PROGRAM PRG_LARS_ValidationAsConfirmation_ORG
VAR
	rtrigNewOuterArrived					: R_TRIG;
	bNewOuterIsProccesing				: BOOL;
	tonValidationTimout					: TON;
	bValidationTimeout					: BOOL;
	bValidationTimeoutReset				: BOOL;
	fbTimeoutCounter						: CTU;
	nCount									: INT;
	fbPerformance							: FB_Interval;

	fbOuterValidationCamera				: FB_SCANNER_CameraSelect;
	(*stOuterValidationCameraOptions		: ST_SCANNER_Options := (eScannerType := E_MV_420_FULL, nImageBuffer := 1, nExpectedResp := 2);*)
	fbOuterValidationEvaluation			: FB_SCANNER_Evaluation;

	fbCheckForDuplicateOuterValidation	: FB_OUTER_CheckDuplicateStatus;

	rtrigOuterValidationCameraDone		: R_TRIG;
	bOuterValidationCameraDone			: BOOL;
	bDataReadyForValidation				: BOOL;
	bQAReject								: BOOL;

	sLastImageLableString				: T_OUTER_Barcode;

	fbMoveOuterData						: FB_OUTER_MoveOuterStatus;
	fbCompleteDataFromConfirmation	: FB_OUTER_CompleteDataFromConfirmation;
	fbMETSValidateOuterForReject			: FB_OUTER_ValidateOuterForReject;
	tofValidateOuterDoneForHMI			: TOF;
	fbMasterListUpdate					: FB_OUTER_MasterListUpdate;

	stLastOuterCompleted					: ST_OUTER_Status;
	sLastReadOuterBarcode				: T_OUTER_Barcode;
	sLastReadConfPackCode1				: T_PACK_Barcode;
	nOutersCompleted						: UDINT;
	bDoneInfo								: BOOL;

	rtrigSetOuterValidationOK			: R_TRIG;
	rtrigSetOuterValidationNOK		: R_TRIG;

	rsOuterRejectStation 				: RS;
	rsOuterRejectConfirmation 		: RS;

	rtrigResetValidationStatus			: R_TRIG;

	sRejectCode						: STRING(255);
	fbArchiveInvalidOuters			: FB_OUTER_ArchiveInvalidOuters;
	aReasonForReject					: ARRAY[0..50] OF STRING(255);
	bClearList							: BOOL;

	fbOuterProduced					: FB_KPI_GenericEfficiency;
	fbOuterInspection					: FB_KPI_OutersEfficiency;

	fbOuterLevelCounter				: FB_KPI_OuterLevelCounter;

	fbQARejectCounter				: FB_CTU32;
	fbOuterValidationIndexOK			: FB_CTU32;

	ctuConsecutiveOuterRejects		: CTU;
	nActualCount						: INT;

	stDummyImageData			: ST_SCANNER_ImageData;		(* image data structure *)
	aDistanceCheck				: ARRAY[1..2] OF FB_TimeDistance;
	bResetCTU						: BOOL;
END_VAR
VAR // added by the converter: edge detectors and wires of the graphical bodies
    _w1 : BOOL;
END_VAR

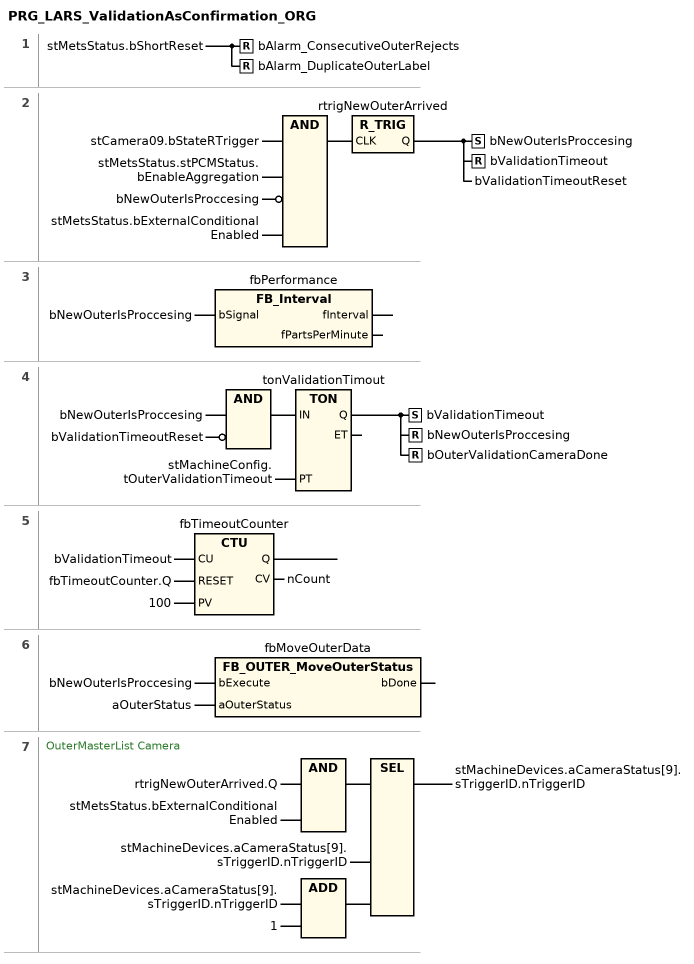
// NETWORK 1
bAlarm_ConsecutiveOuterRejects R= stMetsStatus.bShortReset;
bAlarm_DuplicateOuterLabel R= stMetsStatus.bShortReset;

// NETWORK 2
rtrigNewOuterArrived(CLK := stCamera09.bStateRTrigger AND stMetsStatus.stPCMStatus.bEnableAggregation AND NOT bNewOuterIsProccesing AND stMetsStatus.bExternalConditionalEnabled); // R_TRIG
bNewOuterIsProccesing S= rtrigNewOuterArrived.Q;
bValidationTimeout R= rtrigNewOuterArrived.Q;
bValidationTimeoutReset := rtrigNewOuterArrived.Q;

// NETWORK 3
fbPerformance(bSignal := bNewOuterIsProccesing); // FB_Interval

// NETWORK 4
tonValidationTimout(IN := bNewOuterIsProccesing AND NOT bValidationTimeoutReset, PT := stMachineConfig.tOuterValidationTimeout); // TON
bValidationTimeout S= tonValidationTimout.Q;
bNewOuterIsProccesing R= tonValidationTimout.Q;
bOuterValidationCameraDone R= tonValidationTimout.Q;

// NETWORK 5
fbTimeoutCounter(CU := bValidationTimeout, RESET := fbTimeoutCounter.Q, PV := 100, CV => nCount); // CTU

// NETWORK 6
fbMoveOuterData(bExecute := bNewOuterIsProccesing, aOuterStatus := aOuterStatus); // FB_OUTER_MoveOuterStatus

// NETWORK 7
// OuterMasterList Camera
stMachineDevices.aCameraStatus[9].sTriggerID.nTriggerID := SEL(rtrigNewOuterArrived.Q AND stMetsStatus.bExternalConditionalEnabled, stMachineDevices.aCameraStatus[9].sTriggerID.nTriggerID, stMachineDevices.aCameraStatus[9].sTriggerID.nTriggerID + 1);

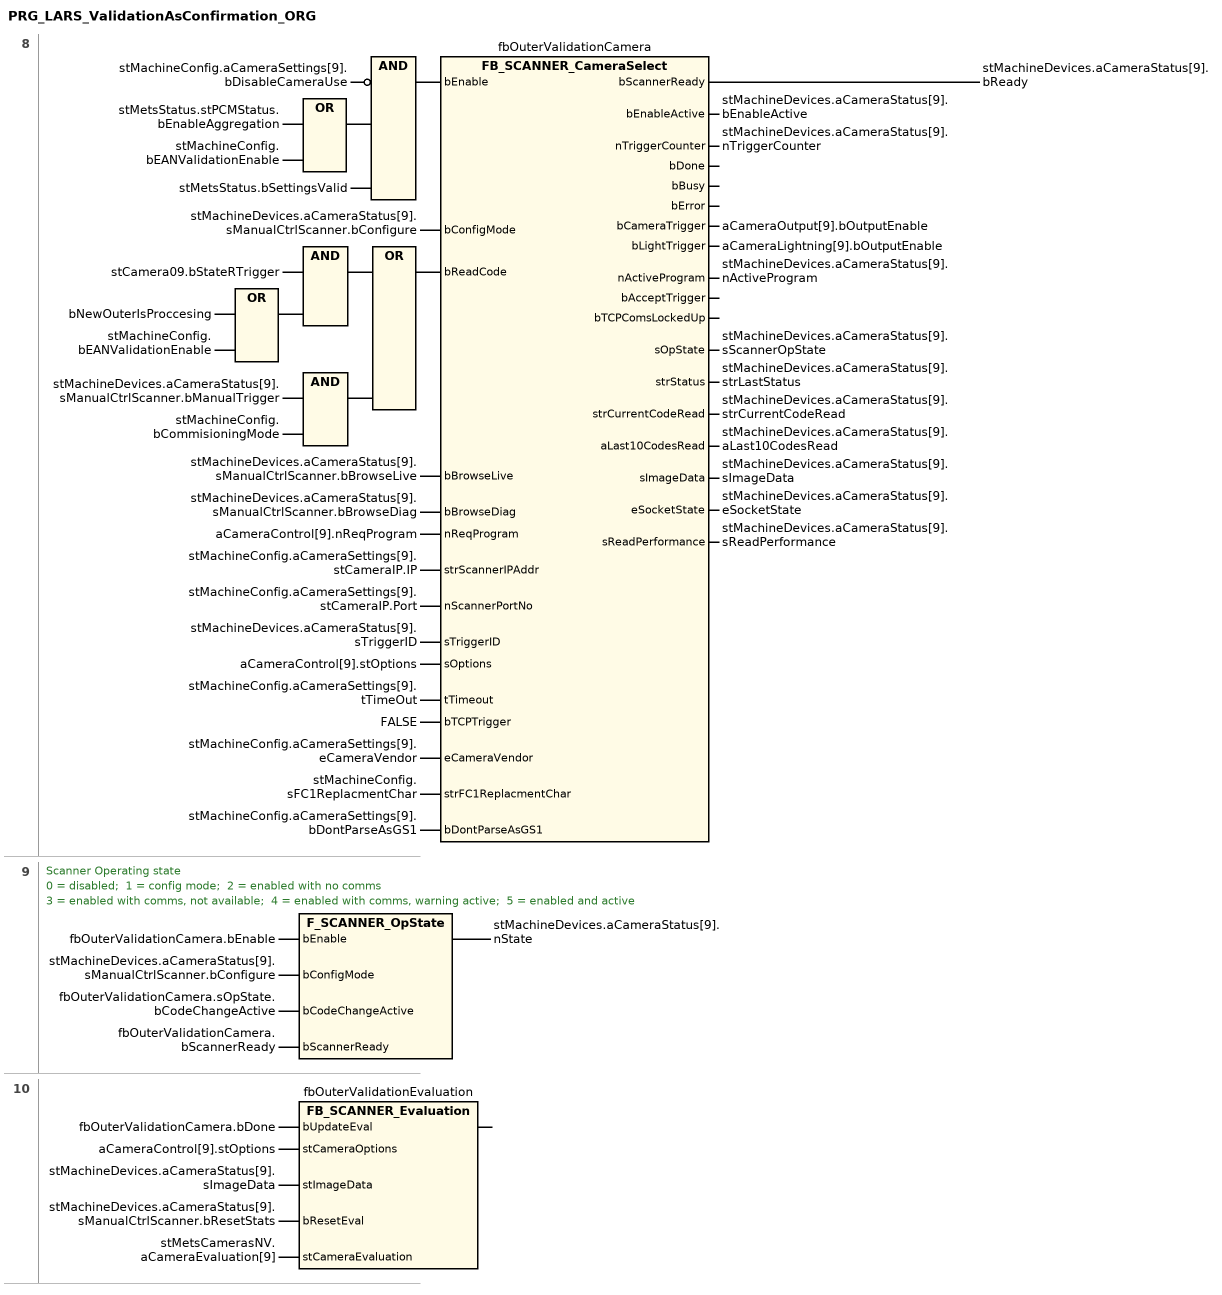
// NETWORK 8
fbOuterValidationCamera(
    bEnable := NOT stMachineConfig.aCameraSettings[9].bDisableCameraUse AND (stMetsStatus.stPCMStatus.bEnableAggregation OR stMachineConfig.bEANValidationEnable) AND stMetsStatus.bSettingsValid,
    bConfigMode := stMachineDevices.aCameraStatus[9].sManualCtrlScanner.bConfigure,
    bReadCode := stCamera09.bStateRTrigger AND (bNewOuterIsProccesing OR stMachineConfig.bEANValidationEnable) OR stMachineDevices.aCameraStatus[9].sManualCtrlScanner.bManualTrigger AND stMachineConfig.bCommisioningMode,
    bBrowseLive := stMachineDevices.aCameraStatus[9].sManualCtrlScanner.bBrowseLive,
    bBrowseDiag := stMachineDevices.aCameraStatus[9].sManualCtrlScanner.bBrowseDiag,
    nReqProgram := aCameraControl[9].nReqProgram,
    strScannerIPAddr := stMachineConfig.aCameraSettings[9].stCameraIP.IP,
    nScannerPortNo := stMachineConfig.aCameraSettings[9].stCameraIP.Port,
    sTriggerID := stMachineDevices.aCameraStatus[9].sTriggerID,
    sOptions := aCameraControl[9].stOptions,
    tTimeout := stMachineConfig.aCameraSettings[9].tTimeOut,
    bTCPTrigger := FALSE,
    eCameraVendor := stMachineConfig.aCameraSettings[9].eCameraVendor,
    strFC1ReplacmentChar := stMachineConfig.sFC1ReplacmentChar,
    bDontParseAsGS1 := stMachineConfig.aCameraSettings[9].bDontParseAsGS1,
    bEnableActive => stMachineDevices.aCameraStatus[9].bEnableActive,
    nTriggerCounter => stMachineDevices.aCameraStatus[9].nTriggerCounter,
    bCameraTrigger => aCameraOutput[9].bOutputEnable,
    bLightTrigger => aCameraLightning[9].bOutputEnable,
    nActiveProgram => stMachineDevices.aCameraStatus[9].nActiveProgram,
    sOpState => stMachineDevices.aCameraStatus[9].sScannerOpState,
    strStatus => stMachineDevices.aCameraStatus[9].strLastStatus,
    strCurrentCodeRead => stMachineDevices.aCameraStatus[9].strCurrentCodeRead,
    aLast10CodesRead => stMachineDevices.aCameraStatus[9].aLast10CodesRead,
    sImageData => stMachineDevices.aCameraStatus[9].sImageData,
    eSocketState => stMachineDevices.aCameraStatus[9].eSocketState,
    sReadPerformance => stMachineDevices.aCameraStatus[9].sReadPerformance); // FB_SCANNER_CameraSelect
stMachineDevices.aCameraStatus[9].bReady := fbOuterValidationCamera.bScannerReady;

// NETWORK 9
// 					Scanner Operating state
// 0 = disabled;  1 = config mode;  2 = enabled with no comms
// 3 = enabled with comms, not available;  4 = enabled with comms, warning active;  5 = enabled and active
//
stMachineDevices.aCameraStatus[9].nState := F_SCANNER_OpState(bEnable := fbOuterValidationCamera.bEnable, bConfigMode := stMachineDevices.aCameraStatus[9].sManualCtrlScanner.bConfigure, bCodeChangeActive := fbOuterValidationCamera.sOpState.bCodeChangeActive, bScannerReady := fbOuterValidationCamera.bScannerReady);

// NETWORK 10
fbOuterValidationEvaluation(
    bUpdateEval := fbOuterValidationCamera.bDone,
    stCameraOptions := aCameraControl[9].stOptions,
    stImageData := stMachineDevices.aCameraStatus[9].sImageData,
    bResetEval := stMachineDevices.aCameraStatus[9].sManualCtrlScanner.bResetStats,
    stCameraEvaluation := stMetsCamerasNV.aCameraEvaluation[9]); // FB_SCANNER_Evaluation

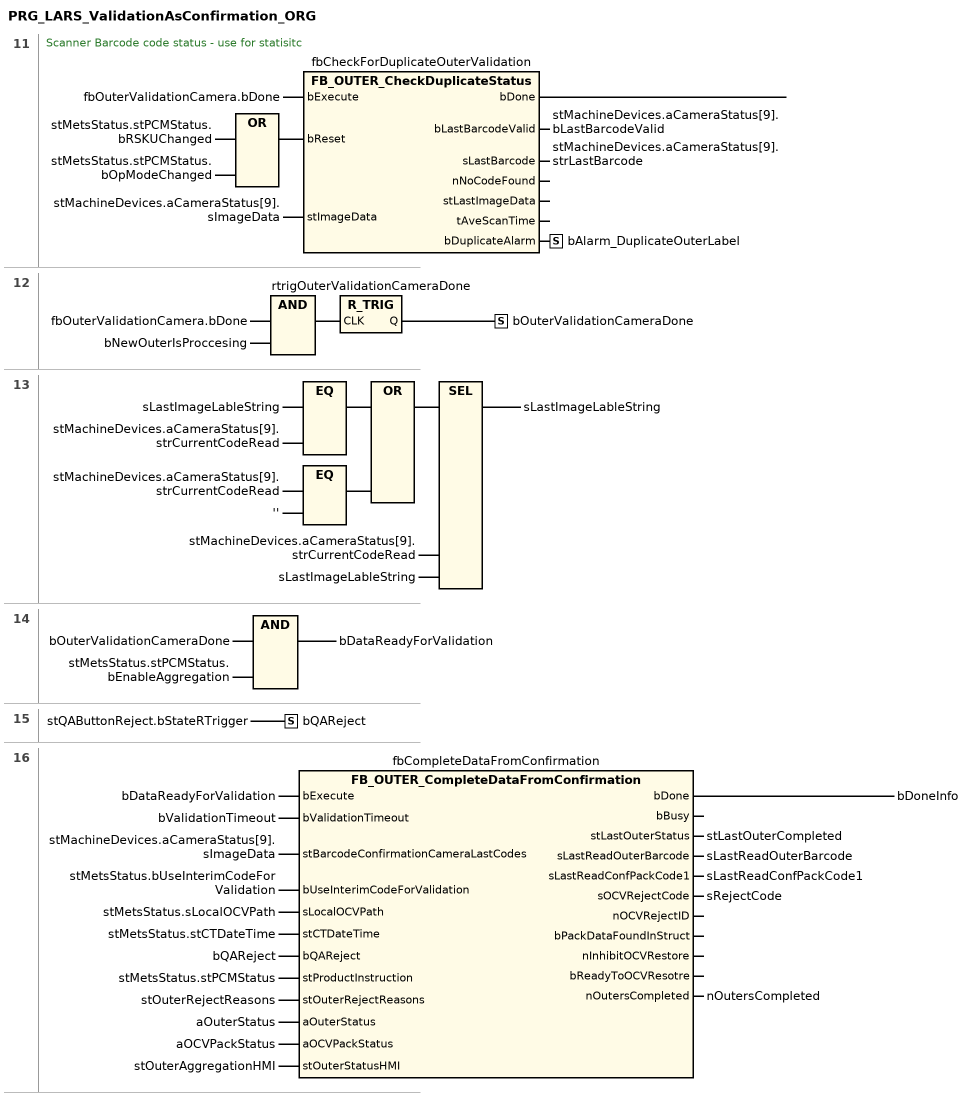
// NETWORK 11
// Scanner Barcode code status - use for statisitc
fbCheckForDuplicateOuterValidation(
    bExecute := fbOuterValidationCamera.bDone,
    bReset := stMetsStatus.stPCMStatus.bRSKUChanged OR stMetsStatus.stPCMStatus.bOpModeChanged,
    stImageData := stMachineDevices.aCameraStatus[9].sImageData,
    bLastBarcodeValid => stMachineDevices.aCameraStatus[9].bLastBarcodeValid,
    sLastBarcode => stMachineDevices.aCameraStatus[9].strLastBarcode); // FB_OUTER_CheckDuplicateStatus
bAlarm_DuplicateOuterLabel S= fbCheckForDuplicateOuterValidation.bDuplicateAlarm;

// NETWORK 12
rtrigOuterValidationCameraDone(CLK := fbOuterValidationCamera.bDone AND bNewOuterIsProccesing); // R_TRIG
bOuterValidationCameraDone S= rtrigOuterValidationCameraDone.Q;

// NETWORK 13
sLastImageLableString := SEL(sLastImageLableString = stMachineDevices.aCameraStatus[9].strCurrentCodeRead OR stMachineDevices.aCameraStatus[9].strCurrentCodeRead = '', stMachineDevices.aCameraStatus[9].strCurrentCodeRead, sLastImageLableString);

// NETWORK 14
bDataReadyForValidation := bOuterValidationCameraDone AND stMetsStatus.stPCMStatus.bEnableAggregation;

// NETWORK 15
bQAReject S= stQAButtonReject.bStateRTrigger;

// NETWORK 16
fbCompleteDataFromConfirmation(
    bExecute := bDataReadyForValidation,
    bValidationTimeout := bValidationTimeout,
    stBarcodeConfirmationCameraLastCodes := stMachineDevices.aCameraStatus[9].sImageData,
    bUseInterimCodeForValidation := stMetsStatus.bUseInterimCodeForValidation,
    sLocalOCVPath := stMetsStatus.sLocalOCVPath,
    stCTDateTime := stMetsStatus.stCTDateTime,
    bQAReject := bQAReject,
    stProductInstruction := stMetsStatus.stPCMStatus,
    stOuterRejectReasons := stOuterRejectReasons,
    aOuterStatus := aOuterStatus,
    aOCVPackStatus := aOCVPackStatus,
    stOuterStatusHMI := stOuterAggregationHMI,
    stLastOuterStatus => stLastOuterCompleted,
    sLastReadOuterBarcode => sLastReadOuterBarcode,
    sLastReadConfPackCode1 => sLastReadConfPackCode1,
    sOCVRejectCode => sRejectCode,
    nOutersCompleted => nOutersCompleted); // FB_OUTER_CompleteDataFromConfirmation
bDoneInfo := fbCompleteDataFromConfirmation.bDone;

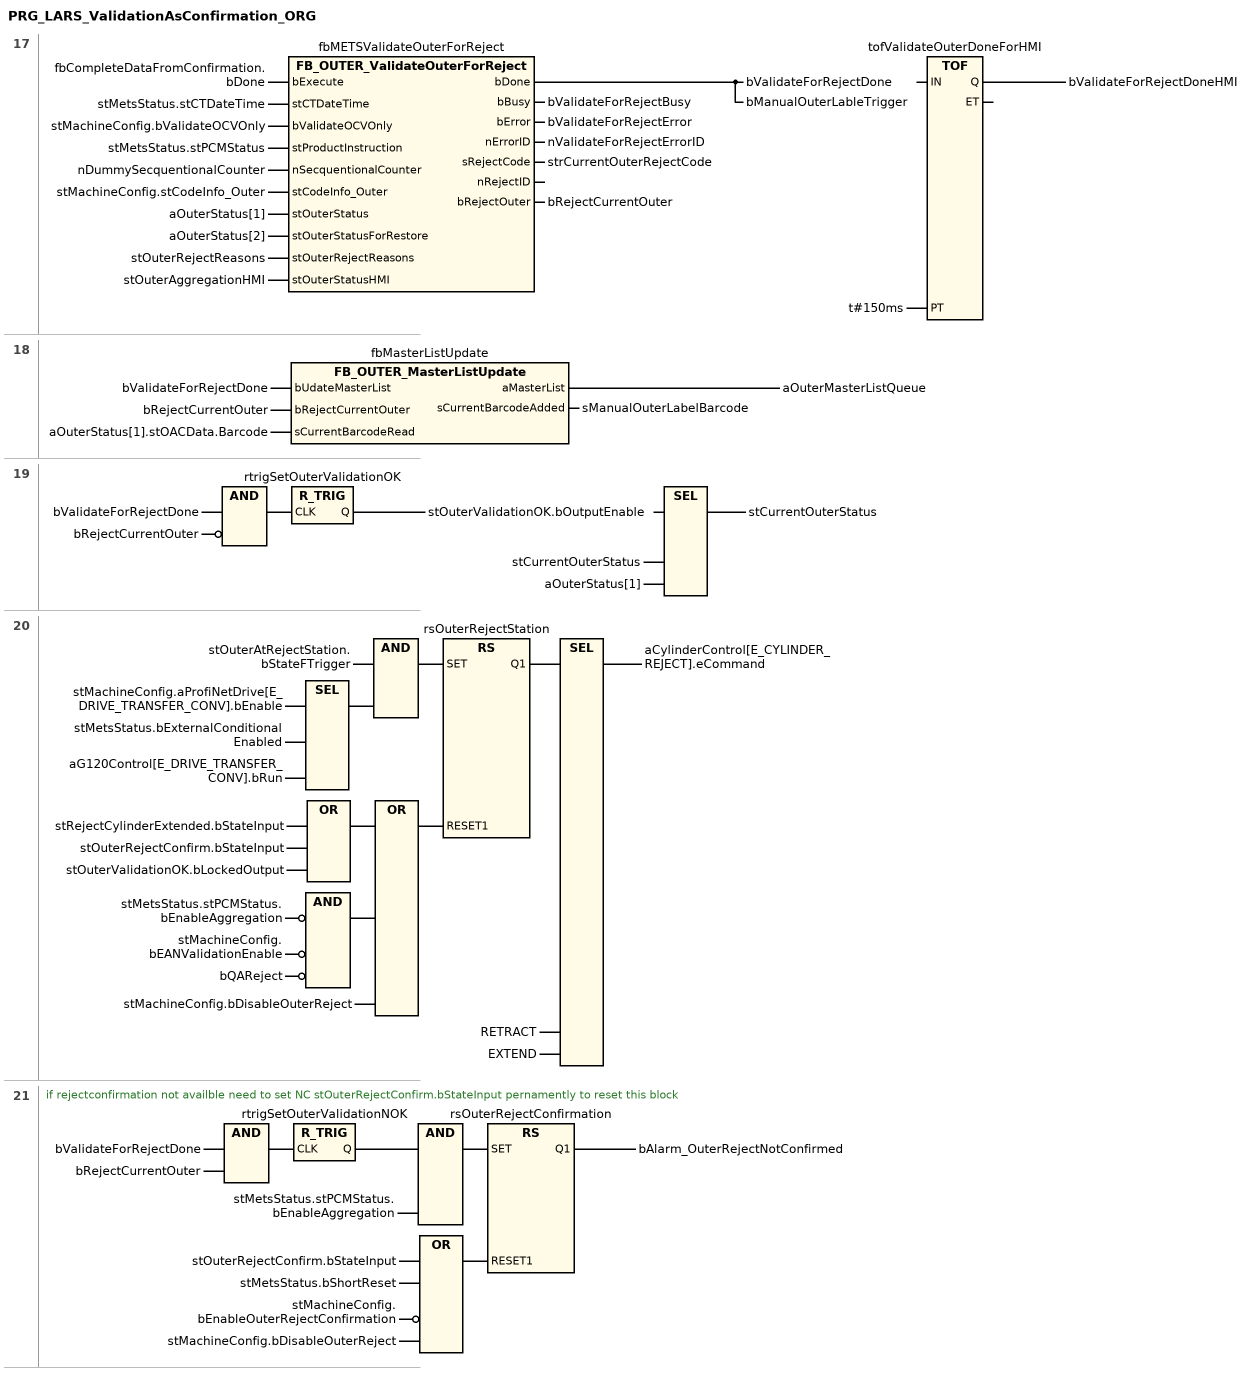
// NETWORK 17
fbMETSValidateOuterForReject(
    bExecute := fbCompleteDataFromConfirmation.bDone,
    stCTDateTime := stMetsStatus.stCTDateTime,
    bValidateOCVOnly := stMachineConfig.bValidateOCVOnly,
    stProductInstruction := stMetsStatus.stPCMStatus,
    nSecquentionalCounter := nDummySecquentionalCounter,
    stCodeInfo_Outer := stMachineConfig.stCodeInfo_Outer,
    stOuterStatus := aOuterStatus[1],
    stOuterStatusForRestore := aOuterStatus[2],
    stOuterRejectReasons := stOuterRejectReasons,
    stOuterStatusHMI := stOuterAggregationHMI,
    bBusy => bValidateForRejectBusy,
    bError => bValidateForRejectError,
    nErrorID => nValidateForRejectErrorID,
    sRejectCode => strCurrentOuterRejectCode,
    bRejectOuter => bRejectCurrentOuter); // FB_OUTER_ValidateOuterForReject
bValidateForRejectDone := fbMETSValidateOuterForReject.bDone;
bManualOuterLableTrigger := fbMETSValidateOuterForReject.bDone;
tofValidateOuterDoneForHMI(IN := fbMETSValidateOuterForReject.bDone, PT := t#150ms); // TOF
bValidateForRejectDoneHMI := tofValidateOuterDoneForHMI.Q;

// NETWORK 18
fbMasterListUpdate(
    bUdateMasterList := bValidateForRejectDone,
    bRejectCurrentOuter := bRejectCurrentOuter,
    sCurrentBarcodeRead := aOuterStatus[1].stOACData.Barcode,
    sCurrentBarcodeAdded => sManualOuterLabelBarcode); // FB_OUTER_MasterListUpdate
aOuterMasterListQueue := fbMasterListUpdate.aMasterList;

// NETWORK 19
rtrigSetOuterValidationOK(CLK := bValidateForRejectDone AND NOT bRejectCurrentOuter); // R_TRIG
stOuterValidationOK.bOutputEnable := rtrigSetOuterValidationOK.Q;
stCurrentOuterStatus := SEL(rtrigSetOuterValidationOK.Q, stCurrentOuterStatus, aOuterStatus[1]);

// NETWORK 20
rsOuterRejectStation(SET := stOuterAtRejectStation.bStateFTrigger AND SEL(stMachineConfig.aProfiNetDrive[E_DRIVE_TRANSFER_CONV].bEnable, stMetsStatus.bExternalConditionalEnabled, aG120Control[E_DRIVE_TRANSFER_CONV].bRun), RESET1 := (stRejectCylinderExtended.bStateInput OR stOuterRejectConfirm.bStateInput OR stOuterValidationOK.bLockedOutput) OR NOT stMetsStatus.stPCMStatus.bEnableAggregation AND NOT stMachineConfig.bEANValidationEnable AND NOT bQAReject OR stMachineConfig.bDisableOuterReject); // RS
aCylinderControl[E_CYLINDER_REJECT].eCommand := SEL(rsOuterRejectStation.Q1, RETRACT, EXTEND);

// NETWORK 21
// if rejectconfirmation not availble need to set NC stOuterRejectConfirm.bStateInput pernamently to reset this block
rtrigSetOuterValidationNOK(CLK := bValidateForRejectDone AND bRejectCurrentOuter); // R_TRIG
rsOuterRejectConfirmation(SET := rtrigSetOuterValidationNOK.Q AND stMetsStatus.stPCMStatus.bEnableAggregation, RESET1 := stOuterRejectConfirm.bStateInput OR stMetsStatus.bShortReset OR NOT stMachineConfig.bEnableOuterRejectConfirmation OR stMachineConfig.bDisableOuterReject); // RS
bAlarm_OuterRejectNotConfirmed := rsOuterRejectConfirmation.Q1;

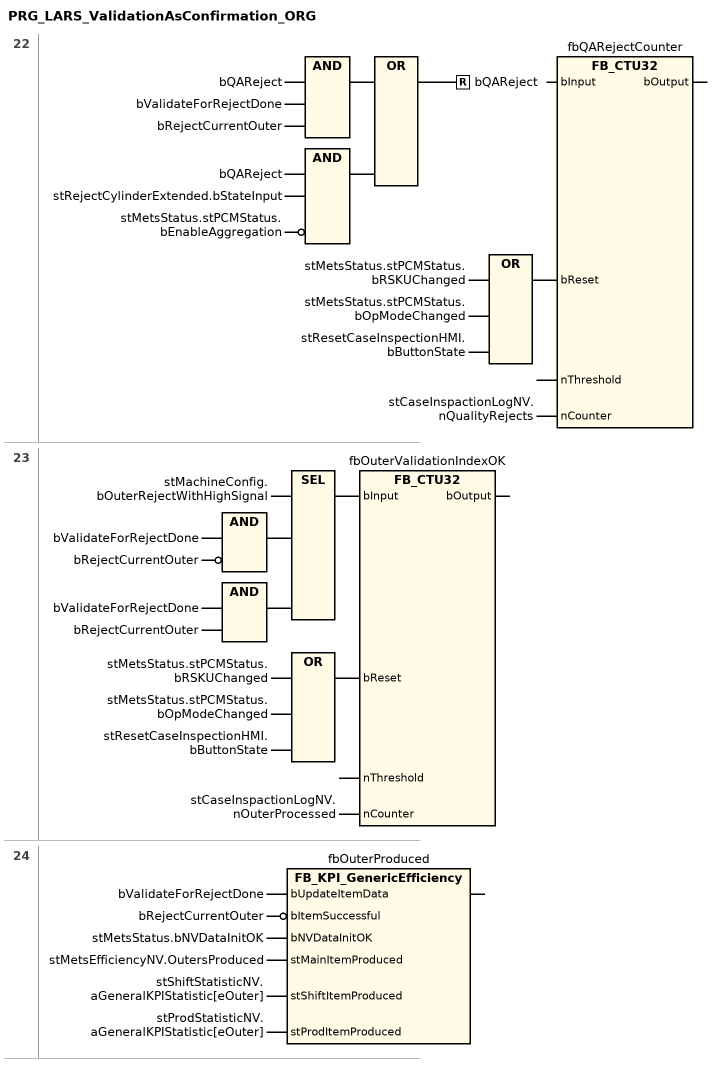
// NETWORK 22
_w1 := bQAReject AND bValidateForRejectDone AND bRejectCurrentOuter OR bQAReject AND stRejectCylinderExtended.bStateInput AND NOT stMetsStatus.stPCMStatus.bEnableAggregation;
bQAReject R= _w1;
fbQARejectCounter(
    bInput := _w1,
    bReset := stMetsStatus.stPCMStatus.bRSKUChanged OR stMetsStatus.stPCMStatus.bOpModeChanged OR stResetCaseInspectionHMI.bButtonState,
    nCounter := stCaseInspactionLogNV.nQualityRejects); // FB_CTU32

// NETWORK 23
fbOuterValidationIndexOK(
    bInput := SEL(stMachineConfig.bOuterRejectWithHighSignal, bValidateForRejectDone AND NOT bRejectCurrentOuter, bValidateForRejectDone AND bRejectCurrentOuter),
    bReset := stMetsStatus.stPCMStatus.bRSKUChanged OR stMetsStatus.stPCMStatus.bOpModeChanged OR stResetCaseInspectionHMI.bButtonState,
    nCounter := stCaseInspactionLogNV.nOuterProcessed); // FB_CTU32

// NETWORK 24
fbOuterProduced(
    bUpdateItemData := bValidateForRejectDone,
    bItemSuccessful := NOT bRejectCurrentOuter,
    bNVDataInitOK := stMetsStatus.bNVDataInitOK,
    stMainItemProduced := stMetsEfficiencyNV.OutersProduced,
    stShiftItemProduced := stShiftStatisticNV.aGeneralKPIStatistic[eOuter],
    stProdItemProduced := stProdStatisticNV.aGeneralKPIStatistic[eOuter]); // FB_KPI_GenericEfficiency

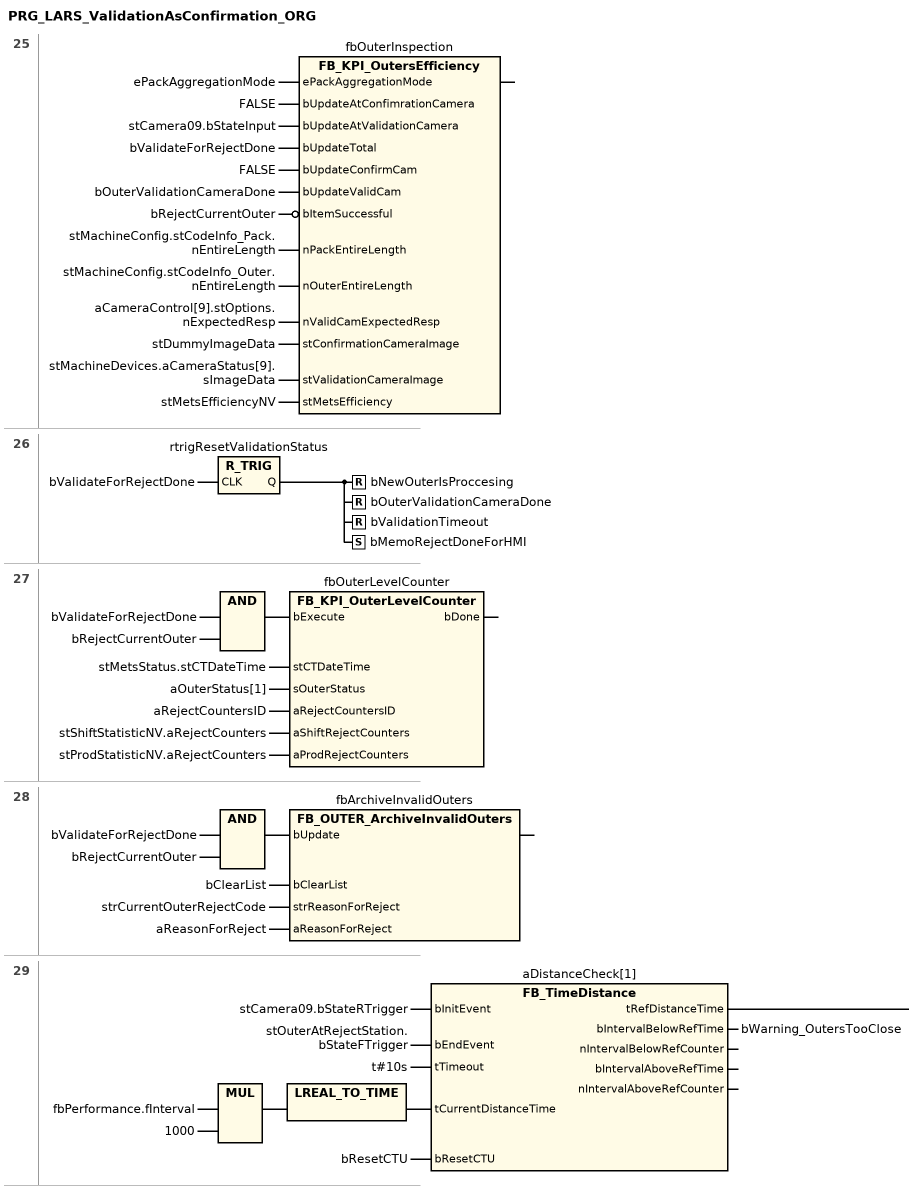
// NETWORK 25
fbOuterInspection(
    ePackAggregationMode := ePackAggregationMode,
    bUpdateAtConfimrationCamera := FALSE,
    bUpdateAtValidationCamera := stCamera09.bStateInput,
    bUpdateTotal := bValidateForRejectDone,
    bUpdateConfirmCam := FALSE,
    bUpdateValidCam := bOuterValidationCameraDone,
    bItemSuccessful := NOT bRejectCurrentOuter,
    nPackEntireLength := stMachineConfig.stCodeInfo_Pack.nEntireLength,
    nOuterEntireLength := stMachineConfig.stCodeInfo_Outer.nEntireLength,
    nValidCamExpectedResp := aCameraControl[9].stOptions.nExpectedResp,
    stConfirmationCameraImage := stDummyImageData,
    stValidationCameraImage := stMachineDevices.aCameraStatus[9].sImageData,
    stMetsEfficiency := stMetsEfficiencyNV); // FB_KPI_OutersEfficiency

// NETWORK 26
rtrigResetValidationStatus(CLK := bValidateForRejectDone); // R_TRIG
bNewOuterIsProccesing R= rtrigResetValidationStatus.Q;
bOuterValidationCameraDone R= rtrigResetValidationStatus.Q;
bValidationTimeout R= rtrigResetValidationStatus.Q;
bMemoRejectDoneForHMI S= rtrigResetValidationStatus.Q;

// NETWORK 27
fbOuterLevelCounter(
    bExecute := bValidateForRejectDone AND bRejectCurrentOuter,
    stCTDateTime := stMetsStatus.stCTDateTime,
    sOuterStatus := aOuterStatus[1],
    aRejectCountersID := aRejectCountersID,
    aShiftRejectCounters := stShiftStatisticNV.aRejectCounters,
    aProdRejectCounters := stProdStatisticNV.aRejectCounters); // FB_KPI_OuterLevelCounter

// NETWORK 28
fbArchiveInvalidOuters(
    bUpdate := bValidateForRejectDone AND bRejectCurrentOuter,
    bClearList := bClearList,
    strReasonForReject := strCurrentOuterRejectCode,
    aReasonForReject := aReasonForReject); // FB_OUTER_ArchiveInvalidOuters

// NETWORK 29
aDistanceCheck[1](
    bInitEvent := stCamera09.bStateRTrigger,
    bEndEvent := stOuterAtRejectStation.bStateFTrigger,
    tTimeout := t#10s,
    tCurrentDistanceTime := LREAL_TO_TIME(fbPerformance.fInterval * 1000),
    bResetCTU := bResetCTU,
    bIntervalBelowRefTime => bWarning_OutersTooClose); // FB_TimeDistance

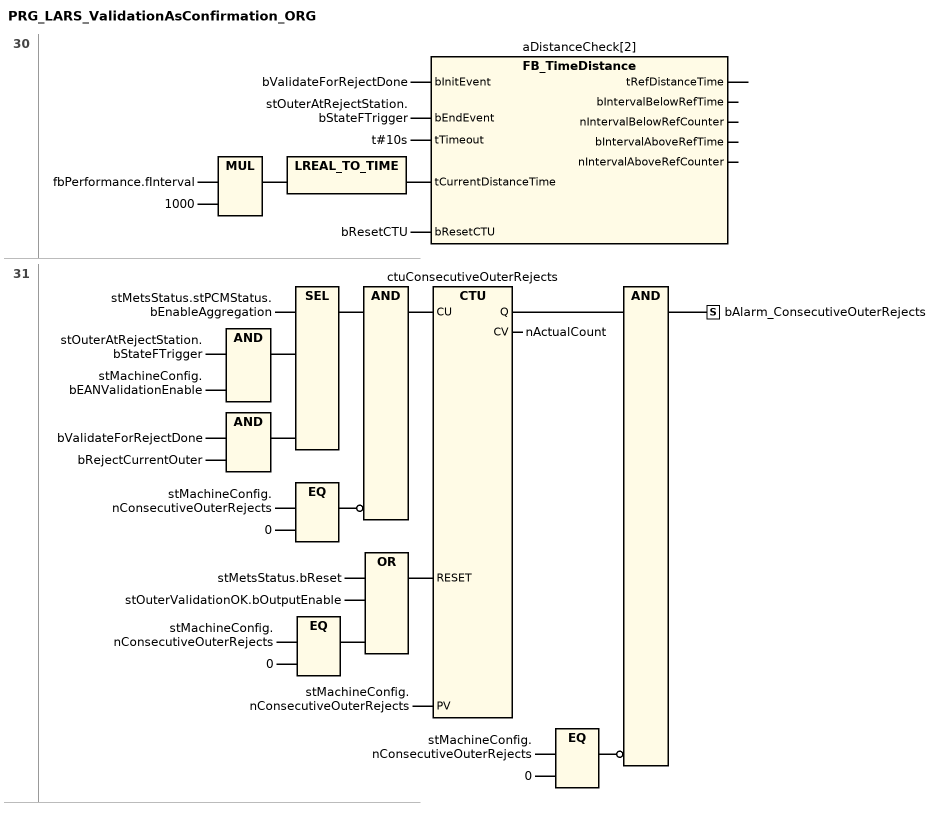
// NETWORK 30
aDistanceCheck[2](
    bInitEvent := bValidateForRejectDone,
    bEndEvent := stOuterAtRejectStation.bStateFTrigger,
    tTimeout := t#10s,
    tCurrentDistanceTime := LREAL_TO_TIME(fbPerformance.fInterval * 1000),
    bResetCTU := bResetCTU); // FB_TimeDistance

// NETWORK 31
ctuConsecutiveOuterRejects(
    CU := SEL(stMetsStatus.stPCMStatus.bEnableAggregation, stOuterAtRejectStation.bStateFTrigger AND stMachineConfig.bEANValidationEnable, bValidateForRejectDone AND bRejectCurrentOuter) AND NOT (stMachineConfig.nConsecutiveOuterRejects = 0),
    RESET := stMetsStatus.bReset OR stOuterValidationOK.bOutputEnable OR stMachineConfig.nConsecutiveOuterRejects = 0,
    PV := stMachineConfig.nConsecutiveOuterRejects,
    CV => nActualCount); // CTU
bAlarm_ConsecutiveOuterRejects S= ctuConsecutiveOuterRejects.Q AND NOT (stMachineConfig.nConsecutiveOuterRejects = 0);

END_PROGRAM

(* stored: Version 1.1.0.1, ProductVersion 3.1.4024.15
   POU PRG_LARS_ValidationAsConfirmation_ORG: Id {54e5a08a-1360-460e-b159-9599c23f94a3}, SpecialFunc None *)
